// TIA Portal project "比赛3" (V15)

(* hardware
DEVICE "S7-1200 station_1"  S7-1200 Station
   slot 0: "Rack_0"  S7-1200 Rack  Rack  V1.0
   slot 1: "PLC_1"  CPU 1215C DC/DC/Rly  6ES7 215-1HG40-0XB0  V4.2
   slot 2: "DI 16x24VDC/DQ 16xRelay_1"  SM 1223 DI16/DQ16 x relay  6ES7 223-1PL32-0XB0  V2.0
   slot 3: "DI 16x24VDC_2"  6ES7 221-1BH32-0XB0  V2.0
   slot 4: "DI 16x24VDC_1"  6ES7 221-1BH32-0XB0  V2.0
DEVICE "HMI_1"  TP900 Comfort
   slot 0: "HMI_1"  TP900 Comfort  6AV2 124-0JC01-0AX0  15.0.0.0
   slot 1: "HMI_RT_1"  TP900 Comfort  6AV2 124-0JC01-0AX0  15.0.0.0
   slot 5: "HMI_1.IE_CP_1"  PROFINET Interface  15.0.0.0
      slot 1: "PROFINET Interface_1"  PROFINET Interface
         slot 1: "Port_1"  Port
         slot 2: "Port_2"  Port
   slot 7: "HMI_1.MPI/DP_CP_1"  MPI/DP Interface  15.0.0.0
*)

// ===== PLC "PLC_1"  CPU 1215C DC/DC/Rly =====

VAR_GLOBAL   // PLC tag table "变量表_1"
   "DI车床准备信号" AT %I2.0 : Bool;
   "DI车床取放工件原点信号" AT %I2.1 : Bool;
   "DI车床运行信号" AT %I2.2 : Bool;
   "DI车床加工完成信号" AT %I2.3 : Bool;
   "DI车床异常信号" AT %I2.4 : Bool;
   "DI车床卡盘松开信号" AT %I2.5 : Bool;
   "DI车床卡盘夹紧信号" AT %I2.6 : Bool;
   "DI车床防护门开门到位信号" AT %I2.7 : Bool;
   "DI加工中心准备信号" AT %I3.0 : Bool;
   "DI加工中心取放工件原点信号" AT %I3.1 : Bool;
   "DI加工中心运行信号" AT %I3.2 : Bool;
   "DI加工中心加工完成信号" AT %I3.3 : Bool;
   "DI加工中心异常信号" AT %I3.4 : Bool;
   "D加工中心平口钳松开信号" AT %I3.5 : Bool;
   "DI加工中心平口钳夹紧信号" AT %I3.6 : Bool;
   "D加工中心防护门开门到位信号" AT %I3.7 : Bool;
   "急停旋钮" AT %I0.0 : Bool;
   "单机联网旋钮" AT %I0.1 : Bool;
   "仓库急停旋钮" AT %I0.2 : Bool;
   "复位按钮" AT %I0.3 : Bool;
   "功能按钮" AT %I0.4 : Bool;
   "启动按钮" AT %I0.5 : Bool;
   "暂停按钮" AT %I0.6 : Bool;
   "加工中心在线测量信号" AT %I0.7 : Bool;
   "仓库解锁按钮" AT %I1.0 : Bool;
   "防护门信号1（光电）" AT %I1.1 : Bool;
   "防护门信号2（光电）" AT %I1.2 : Bool;
   "快换夹具1（方形）" AT %I1.3 : Bool;
   "快换夹具2（大圆形）" AT %I1.4 : Bool;
   "快换夹具3（小圆形）" AT %I1.5 : Bool;
   "运行指示灯" AT %Q0.0 : Bool;
   "车床摄像头清洗" AT %Q0.1 : Bool;
   "铣床摄像头清洗" AT %Q0.2 : Bool;
   "报警指示" AT %Q0.3 : Bool;
   "复位指示灯" AT %Q0.4 : Bool;
   "仓库电磁锁" AT %Q0.5 : Bool;
   "机器人安全信号继电器" AT %Q0.6 : Bool;
   "仓库解锁指示" AT %Q0.7 : Bool;
   "仓库运行指示" AT %Q1.0 : Bool;
   "联网指示" AT %Q1.1 : Bool;
   "DO车床联机信号" AT %Q2.0 : Bool;
   "DO车床启动信号" AT %Q2.1 : Bool;
   "DO车床确认完成信号" AT %Q2.2 : Bool;
   "DO车床程序选择1（8421）" AT %Q2.3 : Bool;
   "DO车床程序选择2（8421）" AT %Q2.4 : Bool;
   "DO车床卡盘控制信号" AT %Q2.5 : Bool;
   "DO车床防护门控制信号" AT %Q2.6 : Bool;
   "DO车床暂停信号" AT %Q2.7 : Bool;
   "DO加工中心联机信号" AT %Q3.0 : Bool;
   "DO加工中心启动信号" AT %Q3.1 : Bool;
   "DO加工中心确认完成信号" AT %Q3.2 : Bool;
   "DO加工中心程序选择1（8421）" AT %Q3.3 : Bool;
   "DO加工中心程序选择2（8421）" AT %Q3.4 : Bool;
   "DO加工中心平口钳控制" AT %Q3.5 : Bool;
   "DO加工中心防护门控制" AT %Q3.6 : Bool;
   "DO加工中心暂停信号" AT %Q3.7 : Bool;
   "车床安全门控制" AT %M5.4 : Bool;
   "CNC安全门控制" AT %M5.5 : Bool;
   "卡盘控制" AT %M5.6 : Bool;
   "平口钳控制" AT %M5.7 : Bool;
   "车床安全门到位信号" AT %M4.4 : Bool;
   "CNC安全门到位信号" AT %M4.5 : Bool;
   "卡盘夹紧信号" AT %M4.6 : Bool;
   "平口钳夹紧信号" AT %M4.7 : Bool;
   "吹气" AT %Q1.2 : Bool;
   "吹气控制" AT %M4.3 : Bool;
   "吹气1" AT %M4.2 : Bool;
END_VAR

DATA_BLOCK "机器人通讯_DB"   // DB2
{ S7_Optimized_Access := 'TRUE' }
VERSION : 0.1
// stored: InstanceOfName 机器人通讯
"机器人通讯"
BEGIN
END_DATA_BLOCK

DATA_BLOCK "robot"   // DB3
{ S7_Optimized_Access := 'FALSE' }
VERSION : 0.1
   VAR
      connect : TCON_IP_v4;
      "40000" : Int;
      "40001" : Int;
      "40002" : Int;
      "40003" : Int;
      "40004" : Int;
      "40005" : Int;
      "40006" : Int;
      "40007X" : Int;
      "40008Y" : Int;
      "40009Z" : Int;
      "40010A" : Int;
      "40011B" : Int;
      "40012C" : Int;
      "40013A1" : Int;
      "40014A2" : Int;
      "40015A3" : Int;
      "40016A4" : Int;
      "40017A5" : Int;
      "40018A6" : Int;
      "40019" : Int;
      "40020" : Int;
      "40021" : Int;
      "40022" : Int;
      "40023" : Int;
      "40024" : Int;
      "40025" : Int;
      "40026" : Int;
      "40027" : Int;
      "40028" : Int;
      "40029" : Int;
      "40030" : Int;
      "40031" : Int;
      "40032" : Int;
      "40033" : Int;
      "40034" : Int;
      "40035" : Int;
      "40036" : Int;
      "40037" : Int;
      "40038" : Int;
      "40039" : Int;
      "40040" : Int;
      "40041" : Int;
      "40042" : Int;
      "40043" : Int;
      "40044" : Int;
      "40045" : Int;
      "40046" : Int;
      "40047" : Int;
      "40048" : Int;
      "40049" : Int;
      "40050" : Int;
      "40051" : Int;
      "40052" : Int;
      "40053" : Int;
      "40054" : Int;
      "40055" : Int;
      "40056" : Int;
      "40057" : Int;
      "40058" : Int;
      "40059" : Int;
      "40060" : Int;
      "40061" : Int;
      "40062" : Int;
      "40063" : Int;
      "40064" : Int;
      "40065" : Int;
      "40081机器人程序选择" : Int;
      "40082" : Int;
      "40083" : Int;
      "40084" : Int;
      "40085" : Int;
      "40086" : Int;
      "40087" : Int;
      "40088" : Int;
      "40089" : Int;
      "40090" : Int;
      "40091" : Int;
      "40092" : Int;
      "40093" : Int;
      "40094" : Int;
      "40095" : Int;
      "40096" : Int;
      "40097" : Int;
      "40098" : Int;
      "40099" : Int;
      "40100" : Int;
      "40101" : Int;
   END_VAR
BEGIN
   connect.InterfaceId := 64;
   connect.ID := 2;
   connect.ActiveEstablished := 1;
   connect.RemotePort := 502;
   connect.RemoteAddress.ADDR[1] := 192;
   connect.RemoteAddress.ADDR[2] := 168;
   connect.RemoteAddress.ADDR[3] := 8;
   connect.RemoteAddress.ADDR[4] := 103;
END_DATA_BLOCK

FUNCTION_BLOCK "机器人通讯"   // FB1, LAD
{ S7_Optimized_Access := 'TRUE' }
VERSION : 0.1
   VAR
      r_done : Bool;
      r_busy : Bool;
      r_error : Bool;
      r_status : Int;
      w_done : Bool;
      w_busy : Bool;
      w_error : Bool;
      w_status : Int;
   END_VAR
BEGIN

REGION Network 1
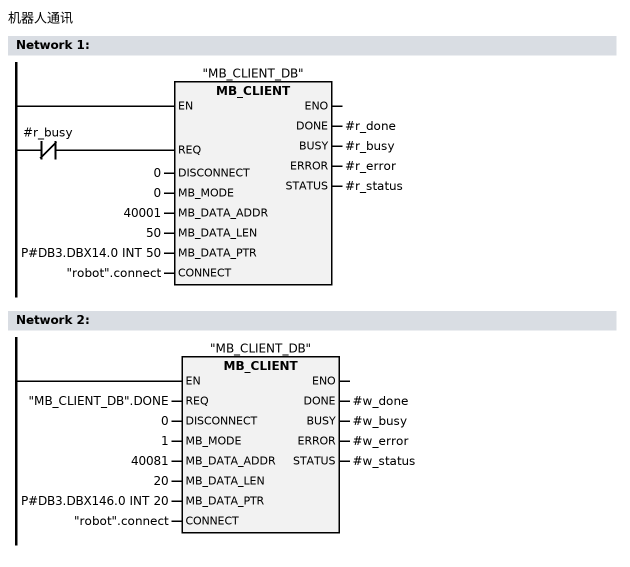
   "MB_CLIENT_DB"(REQ := NOT #r_busy,   // MB_CLIENT
                  DISCONNECT := 0,
                  MB_MODE := 0,
                  MB_DATA_ADDR := 40001,
                  MB_DATA_LEN := 50,
                  MB_DATA_PTR := P#DB3.DBX14.0 INT 50,
                  CONNECT := "robot".connect,
                  DONE => #r_done,
                  BUSY => #r_busy,
                  ERROR => #r_error,
                  STATUS => #r_status);
END_REGION

REGION Network 2
   "MB_CLIENT_DB"(REQ := "MB_CLIENT_DB".DONE,   // MB_CLIENT
                  DISCONNECT := 0,
                  MB_MODE := 1,
                  MB_DATA_ADDR := 40081,
                  MB_DATA_LEN := 20,
                  MB_DATA_PTR := P#DB3.DBX146.0 INT 20,
                  CONNECT := "robot".connect,
                  DONE => #w_done,
                  BUSY => #w_busy,
                  ERROR => #w_error,
                  STATUS => #w_status);
END_REGION
END_FUNCTION_BLOCK

FUNCTION "辅助控制" : Void   // FC1, LAD
{ S7_Optimized_Access := 'TRUE' }
VERSION : 0.1
BEGIN

REGION Network 1
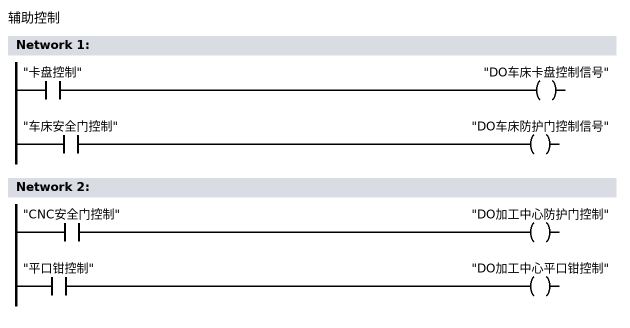
   RUNG wire#powerrail
      Contact( "卡盘控制" )
      Coil( "DO车床卡盘控制信号" )
   END_RUNG
   RUNG wire#powerrail
      Contact( "车床安全门控制" )
      Coil( "DO车床防护门控制信号" )
   END_RUNG
   // the same network as SCL:
   "DO车床卡盘控制信号" := "卡盘控制";
   "DO车床防护门控制信号" := "车床安全门控制";
END_REGION

REGION Network 2
   RUNG wire#powerrail
      Contact( "CNC安全门控制" )
      Coil( "DO加工中心防护门控制" )
   END_RUNG
   RUNG wire#powerrail
      Contact( "平口钳控制" )
      Coil( "DO加工中心平口钳控制" )
   END_RUNG
   // the same network as SCL:
   "DO加工中心防护门控制" := "CNC安全门控制";
   "DO加工中心平口钳控制" := "平口钳控制";
END_REGION
END_FUNCTION

ORGANIZATION_BLOCK "Main"   // OB1, LAD, ProgramCycle
TITLE = "Main Program Sweep (Cycle)"
{ S7_Optimized_Access := 'TRUE' }
VERSION : 0.1
   VAR_INPUT
      Initial_Call : Bool;   // Initial call of this OB
      Remanence : Bool;   // =True, if remanent data are available
   END_VAR
BEGIN

REGION Network 1
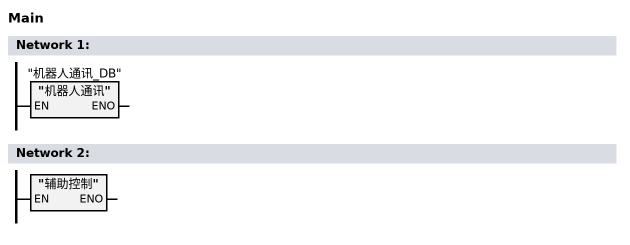
   RUNG wire#powerrail
      "机器人通讯_DB"()
   END_RUNG
   // the same network as SCL:
   "机器人通讯_DB"();   // "机器人通讯"
END_REGION

REGION Network 2
   RUNG wire#powerrail
      "辅助控制"()
   END_RUNG
   // the same network as SCL:
   "辅助控制"();
END_REGION
END_ORGANIZATION_BLOCK

(* ===== HMI "HMI_RT_1" =====
system functions are stored by id; their names below are inferred from use
connection "HMI_连接_1": ETHERNET, S7_1200_OMS

HMI tags "默认变量表"
   "Tag_ScreenNumber" : UInt, internal
   "robot_40081机器人程序选择" : Int = PLC robot.40081机器人程序选择 AT %DB3.DBW146, 1 s
   "robot_40007X" : Int = PLC robot.40007X AT %DB3.DBW28, 1 s
   "robot_40008Y" : Int = PLC robot.40008Y AT %DB3.DBW30, 1 s
   "robot_40009Z" : Int = PLC robot.40009Z AT %DB3.DBW32, 1 s
   "robot_40010A" : Int = PLC robot.40010A AT %DB3.DBW34, 1 s
   "robot_40011B" : Int = PLC robot.40011B AT %DB3.DBW36, 1 s
   "robot_40012C" : Int = PLC robot.40012C AT %DB3.DBW38, 1 s
   "robot_40013A1" : Int = PLC robot.40013A1 AT %DB3.DBW40, 1 s
   "robot_40014A2" : Int = PLC robot.40014A2 AT %DB3.DBW42, 1 s
   "robot_40015A3" : Int = PLC robot.40015A3 AT %DB3.DBW44, 1 s
   "robot_40016A4" : Int = PLC robot.40016A4 AT %DB3.DBW46, 1 s
   "robot_40017A5" : Int = PLC robot.40017A5 AT %DB3.DBW48, 1 s
   "robot_40018A6" : Int = PLC robot.40018A6 AT %DB3.DBW50, 1 s
   "CNC安全门控制" : Bool = PLC CNC安全门控制 AT %M5.5, 1 s
   "CNC安全门到位信号" : Bool = PLC CNC安全门到位信号 AT %M4.5, 1 s
   "DI车床防护门开门到位信号" : Bool = PLC DI车床防护门开门到位信号 AT %I2.7, 1 s
   "车床安全门控制" : Bool = PLC 车床安全门控制 AT %M5.4, 1 s
   "卡盘控制" : Bool = PLC 卡盘控制 AT %M5.6, 1 s
   "DI车床卡盘松开信号" : Bool = PLC DI车床卡盘松开信号 AT %I2.5, 1 s
   "D加工中心平口钳松开信号" : Bool = PLC D加工中心平口钳松开信号 AT %I3.5, 1 s
   "平口钳控制" : Bool = PLC 平口钳控制 AT %M5.7, 1 s
   "吹气控制" : Bool = PLC 吹气控制 AT %M4.3, 1 s
   "吹气" : Bool = PLC 吹气 AT %Q1.2, 1 s
   "robot_40030" : Int = PLC robot.40030 AT %DB3.DBW74, 1 s

screen "画面_1" 800x420
   Button "按钮_1" at 74,69 size 96x32; TextOff '吹气'
      on Press: SetBit("吹气控制")
      on Release: ResetBit("吹气控制")
   Circle "圆_1" at 243,62 size 48x48
      Appearance <- "吹气"
   TextField "文本域_1" at 239,29 size 61x17; Text '吹气指示'

screen "根画面" 800x420, template "Template_1"
   on GenerateScreen: SetTag("Tag_ScreenNumber", 1)
   TextField "HmiScreenItemData" at 80,167 size 640x22; Text 'Text'
   IOField "I/O 域_1" at 141,37 size 96x32; FormatPattern s999
      ProcessValue <- "robot_40081机器人程序选择"
   TextField "文本域_1" at 22,46 size 103x17; Text '机器人程序选择'
   IOField "I/O 域_2" at 44,207 size 82x35; FormatPattern s99999
      ProcessValue <- "robot_40007X"
   IOField "I/O 域_4" at 152,209 size 82x35; FormatPattern s99999
      ProcessValue <- "robot_40008Y"
   IOField "I/O 域_5" at 260,211 size 82x35; FormatPattern s99999
      ProcessValue <- "robot_40009Z"
   IOField "I/O 域_6" at 368,213 size 82x35; FormatPattern s99999
      ProcessValue <- "robot_40010A"
   IOField "I/O 域_7" at 476,215 size 82x35; FormatPattern s99999
      ProcessValue <- "robot_40011B"
   IOField "I/O 域_8" at 584,217 size 82x35; FormatPattern s99999
      ProcessValue <- "robot_40012C"
   IOField "I/O 域_9" at 44,283 size 82x35; FormatPattern s99999
      ProcessValue <- "robot_40013A1"
   IOField "I/O 域_10" at 152,283 size 82x35; FormatPattern s99999
      ProcessValue <- "robot_40014A2"
   IOField "I/O 域_11" at 260,285 size 82x35; FormatPattern s99999
      ProcessValue <- "robot_40015A3"
   IOField "I/O 域_12" at 368,287 size 82x35; FormatPattern s99999
      ProcessValue <- "robot_40016A4"
   IOField "I/O 域_13" at 476,289 size 82x35; FormatPattern s99999
      ProcessValue <- "robot_40017A5"
   IOField "I/O 域_14" at 584,291 size 82x35; FormatPattern s99999
      ProcessValue <- "robot_40018A6"
   TextField "文本域_2" at 75,178 size 19x29; Text 'X'
   TextField "文本域_3" at 184,179 size 19x29; Text 'Y'
   TextField "文本域_4" at 289,181 size 19x29; Text 'Z'
   TextField "文本域_5" at 398,184 size 19x29; Text 'A'
   TextField "文本域_6" at 505,185 size 19x29; Text 'B'
   TextField "文本域_7" at 614,186 size 19x29; Text 'C'
   TextField "文本域_8" at 505,262 size 33x29; Text 'A5'
   TextField "文本域_9" at 614,263 size 33x29; Text 'A6'
   TextField "文本域_10" at 291,261 size 33x29; Text 'A3'
   TextField "文本域_11" at 400,262 size 33x29; Text 'A4'
   TextField "文本域_12" at 77,260 size 33x29; Text 'A1'
   TextField "文本域_13" at 186,260 size 33x29; Text 'A2'
   Button "按钮_1" at 560,40 size 96x32; TextOff 'CNC安全门控制'
      on Press: SetBit("CNC安全门控制")
      on Release: ResetBit("CNC安全门控制")
   Circle "圆_1" at 695,37 size 37x37
      Appearance <- "DI车床防护门开门到位信号"
   Circle "圆_2" at 457,32 size 37x37
      Appearance <- "DI车床防护门开门到位信号"
   Button "按钮_2" at 321,35 size 108x32; TextOff '车床安全门控制'
      on Release: ResetBit("车床安全门控制")
      on Press: SetBit("车床安全门控制")
   Button "按钮_3" at 330,104 size 96x32; TextOff '卡盘控制'
      on Release: ResetBit("卡盘控制")
      on Press: SetBit("卡盘控制")
   Button "按钮_4" at 560,104 size 96x32; TextOff '平口钳控制'
      on Release: ResetBit("平口钳控制")
      on Press: SetBit("平口钳控制")
   Circle "圆_3" at 457,97 size 37x37
      Appearance <- "DI车床卡盘松开信号"
   Circle "圆_4" at 697,104 size 37x37
      Appearance <- "D加工中心平口钳松开信号"
   IOField "I/O 域_3" at 687,293 size 82x35; FormatPattern s99999
      ProcessValue <- "robot_40030"
   TextField "文本域_14" at 701,264 size 33x29; Text 'A7'

Template "Template_1" 800x420
   Button "退出" at 720,360 size 78x58; TextOff '退出'; PictureOff "ExitRuntime_TP900_Comfort_TR"; PictureOn "ExitRuntime_TP900_Comfort_TR"
      on Release: StopRuntime(0)
   Button "Template_Button" at 640,360 size 78x58; TextOff 'Text'
   Button "Template_Button_1" at 560,360 size 78x58; TextOff 'Text'
   Button "Template_Button_2" at 480,360 size 78x58; TextOff 'Text'
   Button "Template_Button_3" at 400,360 size 78x58; TextOff 'Text'
   Button "Template_Button_4" at 321,360 size 78x58; TextOff 'Text'
   Button "Template_Button_5" at 241,360 size 78x58; TextOff 'Text'
   Button "Template_Button_6" at 161,360 size 78x58; TextOff 'Text'
   Button "报警" at 81,360 size 78x58; TextOff '报警'; PictureOff "AlarmDisplay_TP900_Comfort_TR"; PictureOn "AlarmDisplay_TP900_Comfort_TR"
      on Release: function_ef3f5d25("报警窗口_Unacknowledged", -1)
   Button "起始画面" at 1,360 size 78x58; TextOff '起始画面'; PictureOff "NavigateHome_TP900_Comfort_TR"; PictureOn "NavigateHome_TP900_Comfort_TR"
      on Release: ActivateScreen("根画面", 0)
*)